// SIMATIC S7-200 SMART project (STEP 7-Micro/WIN SMART), CPU ST40

SYMBOL_TABLE Table 1
Motor            Q0.0
OFF_Switch       I0.1
Start_Switch     I0.0
Timer            T101
END_SYMBOL_TABLE

ORGANIZATION_BLOCK MAIN:OB1
TITLE=Program Comments
BEGIN
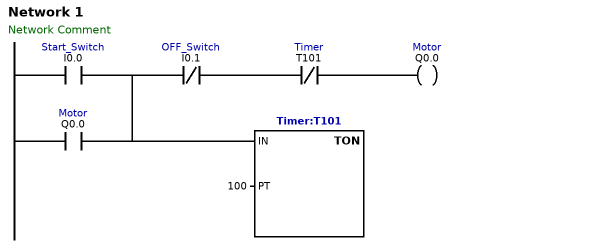
Network 1
// Network Comment
LD     Start_Switch:I0.0
O      Motor:Q0.0
LPS
AN     OFF_Switch:I0.1
AN     Timer:T101
=      Motor:Q0.0
LPP
TON    Timer:T101, 100
END_ORGANIZATION_BLOCK
